// TIA Portal V19 export
DATA_BLOCK "LB111"   // DB25
// stored: InstanceOfName ButtonsSafe_LB111, InstanceOfType FB
"ButtonsSafe_LB111"
   // VAR_INPUT
   //    Reset_OthersPBs_Activation_IN : Bool;
   // END_VAR
   // VAR_OUTPUT
   //    Reset_OthersPBs_Activation_OUT : Bool;
   // END_VAR
   // VAR
   //    i : Int;
   //    iOperation : Int;
   //    iConcurrentOperation : Int;
   //    SettingWriteDone { S7_SetPoint := 'True'} : Bool;
   //    PbPanel { S7_SetPoint := 'True'} : "Buttons2Hands";
   //    PB : Struct
   //       ResetAlarms : Bool;
   //       Coilcar_Up : Bool;
   //       Coilcar_Down : Bool;
   //       Coilcar_Fwd : Bool;
   //       Coilcar_Bwd : Bool;
   //       Jaws_Open : Bool;
   //       Jaws_Close : Bool;
   //       Decoiler_Fwd : Bool;
   //       Decoiler_Bwd : Bool;
   //       SnubberLift_Up : Bool;
   //       SnubberLift_Down : Bool;
   //       SnubberRoll_Fwd : Bool;
   //       SnubberRoll_Bwd : Bool;
   //    END_STRUCT;
   // END_VAR
BEGIN
END_DATA_BLOCK
